// TIA Portal V19 export
DATA_BLOCK "plcStateEvaluation_DB_1"   // DB29
// stored: InstanceOfName plcStateEvaluation, InstanceOfType FB
"plcStateEvaluation"
   // VAR_INPUT
   //    primaryID : Int;
   //    plc1OperationState : UInt;
   //    plc2OperationState : UInt;
   //    plcOperationStateSystem : UInt;
   //    plcMrpRingState : UInt;
   // END_VAR
   // VAR_OUTPUT
   //    PLC_OperateStatus : Int;
   //    PLC_MrpState : Int;
   //    PLC1_LEDStatus : Int;
   //    PLC2_LEDStatus : Int;
   // END_VAR
   // VAR_IN_OUT
   //    PLC12_StopMonitoring : Int;
   // END_VAR
   // VAR
   //    statPrimaryID : Int;
   //    statPlc1State : UInt;
   //    statPlc2State : UInt;
   //    statPlcStateSystem : UInt;
   //    statPlcMrpRingState : UInt;
   //    statPlcStatus : Int;
   //    statPLC12StopMonitoring : Int;
   // END_VAR
BEGIN
END_DATA_BLOCK
